// TIA Portal V20 export
DATA_BLOCK "DB_LoaderOptions"   // DB1305
{ S7_Optimized_Access := 'TRUE' }
AUTHOR : SAN
// stored: AutoNumber false, IsRetainMemResEnabled true, MemoryReserve 20, RetainMemoryReserve 20
   VAR RETAIN
      ExtLoadUnload : Struct
         SeparatePos : Bool;
         CommonPos : Bool;
         Disabled : Bool;
      END_STRUCT;
      Blowing : Struct
         Inside : Bool;
         NearSas : Bool;
         Disabled : Bool;
      END_STRUCT;
      Washing : Struct
         Enabled : Bool;
         Disabled : Bool;
      END_STRUCT;
      PartControl : Struct
         Individual : Bool;
         Common : Bool;
         Disabled : Bool;
         AnalogMeasure : Bool;
         DigitalMeasure : Bool;
      END_STRUCT;
   END_VAR
   VAR
      Stop_Restart : Struct
         BasicVersion : Bool;
      END_STRUCT;
      IntLoadUnload : Struct
         SeparatePos : Bool;
         CommonPos : Bool;
      END_STRUCT;
      BwLoadUnload : Struct
         SeparatePos : Bool;
         CommonPos : Bool;
      END_STRUCT;
      BwControl : Struct
         UndrilledDrilledCtrlSeparate : Bool;
         UndrilledDrilledCtrlCommon : Bool;
         Disabled : Bool;
      END_STRUCT;
      ActPartControlIn : Struct
         Stop : Bool := TRUE;
      END_STRUCT;
      ActPartControlOut : Struct
         Stop : Bool := TRUE;
      END_STRUCT;
      ActBwControlIn : Struct
         Stop : Bool := TRUE;
      END_STRUCT;
      Fixture : Struct
         UnloadingDisabled : Bool;
         LoadingDisabled : Bool;
         BlowingDisabled : Bool;
         ReleaseDisabled : Bool;
         V_InitDisabled : Bool;
         W_InitDisabled : Bool;
      END_STRUCT;
   END_VAR
BEGIN
END_DATA_BLOCK
